// TwinCAT 3 PLC project MAIN
// ProgramVersion: 3.1.4024.0
// libraries:
//   Tc2_Standard, * (Beckhoff Automation GmbH)
//   Tc2_System, * (Beckhoff Automation GmbH)
//   Tc3_Module, * (Beckhoff Automation GmbH)
// project tree:
//   / PlcTask.TcTTO
//   POUs/ MAIN.TcPOU
// real-time tasks:
//   TASK PlcTask: cycle T#10ms, priority 20, ADS port 350
//   TASK PlcTask1: cycle T#10ms, priority 21, ADS port 351
// I/O:
//   DEVICE Device 1 (EtherCAT), AmsNetId 172.18.64.1.2.1
//     Term 1 (EK1100) [EK1100 EtherCAT Coupler (2A E-Bus)]
//       Term 2 (EL1008) [EL1008 8Ch. Dig. Input 24V, 3ms]
//       Term 3 (EL2008) [EL2008 8Ch. Dig. Output 24V, 0.5A]

CONFIGURATION MAIN
    RESOURCE PLC ON TwinCAT3
        TASK PlcTask(INTERVAL := T#10ms, PRIORITY := 21);
        PROGRAM MAIN WITH PlcTask : MAIN;
    END_RESOURCE
END_CONFIGURATION

// ---- POUs/MAIN.TcPOU
PROGRAM MAIN
VAR
    // ===== Inputs (map these in I/O Mapping or force online) =====
    StartBtn    : BOOL;  // Start command (rising edge)
    StopBtn     : BOOL;  // Emergency/stop command (rising edge)
    DepressSw   : BOOL;  // TRUE when forward limit (depressor) is reached
    HomeSw      : BOOL;  // TRUE when returned to home

    // ===== Outputs (map these to your DOs) =====
    MotorFwd    : BOOL;  // Drive forward
    MotorBwd    : BOOL;  // Drive backward

    // ===== Step / control =====
    Step        : INT := 0;    // 0=IDLE, 10=FWD, 20=BWD, 30=DONE
    StartEdge   : R_TRIG;      // Rising-edge detector for StartBtn
    StopEdge    : R_TRIG;      // Rising-edge detector for StopBtn

    // ===== Timer =====
    tMoveTmr    : TON;         // Movement timeout timer
    T_MOVE_MAX  : TIME := T#10S;
END_VAR

// --- Edge detection (call FB instances each cycle) ---
StartEdge(CLK := StartBtn);
StopEdge(CLK := StopBtn);

// --- Global STOP: drop outputs and go idle ---
IF StopEdge.Q THEN
    MotorFwd := FALSE;
    MotorBwd := FALSE;
    Step := 0;
    tMoveTmr(IN := FALSE);
END_IF

CASE Step OF

    0: // IDLE
        MotorFwd := FALSE;
        MotorBwd := FALSE;
        tMoveTmr(IN := FALSE);

        // Start only if not already at forward limit
        IF StartEdge.Q AND NOT DepressSw THEN
            Step := 10;
        END_IF

    10: // MOVE FORWARD until DepressSw or timeout
        MotorFwd := TRUE;
        MotorBwd := FALSE;
        tMoveTmr(IN := TRUE, PT := T_MOVE_MAX);

        IF DepressSw THEN
            MotorFwd := FALSE;
            tMoveTmr(IN := FALSE);
            Step := 20;
        ELSIF tMoveTmr.Q THEN
            MotorFwd := FALSE;
            Step := 0; // timeout -> back to IDLE
        END_IF

    20: // MOVE BACKWARD until HomeSw or timeout
        MotorFwd := FALSE;
        MotorBwd := TRUE;
        tMoveTmr(IN := TRUE, PT := T_MOVE_MAX);

        IF HomeSw THEN
            MotorBwd := FALSE;
            tMoveTmr(IN := FALSE);
            Step := 30;
        ELSIF tMoveTmr.Q THEN
            MotorBwd := FALSE;
            Step := 0; // timeout -> back to IDLE
        END_IF

    30: // DONE → back to IDLE
        MotorFwd := FALSE;
        MotorBwd := FALSE;
        Step := 0;

END_CASE

END_PROGRAM
